// TIA Portal V20 export
TYPE "LER_typeCommunicationConfiguration"
// stored: Access Published
   STRUCT
      disableAlarms : Bool;
      SEND { S7_SetPoint := 'True'} : "LER_typeCommunicationBSENDConfiguration";
      RCV { S7_SetPoint := 'True'} : "LER_typeCommunicationBRCVConfiguration";
   END_STRUCT;
END_TYPE
